{attribute 'qualified_only'}
{attribute 'to_string'}
TYPE E_GROUP_CHECK :
(
  NULL,
  REFERENCE_GROUP_REF_INVALID := 9000,
  REFERENCE_AXIS_REF_INVALID,
  REFERENCE_CTRL_INVALID,
  REFERENCE_STATE_INVALID,
  REFERENCE_MOVER_ITF_INVALID,
  REFERENCE_XPU_INFO_INVALID,

  CHECK_DONE              := 10000
)UINT;
END_TYPE

(* stored: Version 1.1.0.1
   DUT E_GROUP_CHECK: Id {c1a7eb5c-1432-4ebc-9717-a47f59982c80} *)
